// TIA Portal project "SistemaIrrigazione2" (V15.1)

(* hardware
DEVICE "S7-1200 station_1"  S7-1200 Station
   slot 0: "Telaio di montaggio_0"  S7-1200 Rack  Rack  V1.0
   slot 1: "PLC_1"  CPU 1214C DC/DC/DC  6ES7 214-1AG40-0XB0  V4.2
*)

// ===== PLC "PLC_1"  CPU 1214C DC/DC/DC =====

VAR_GLOBAL   // PLC tag table "Tabella delle variabili standard"
   "SEC" AT %I0.0 : Bool;
   "Apri_0" AT %Q0.1 : Bool;
   "Apri_1" AT %Q0.2 : Bool;
   "Apri_2" AT %Q0.3 : Bool;
   "Chiudi_0" AT %Q0.4 : Bool;
   "Chiudi_1" AT %Q0.5 : Bool;
   "Chiudi_2" AT %Q0.6 : Bool;
END_VAR

VAR_GLOBAL CONSTANT   // PLC tag table "Tabella delle variabili standard"
   "IntervalloIrrigazione" : Time := T#5m;
   "DurataApertura" : Time := T#10s;
   "DurataChiusura" : Time := T#10s;
   "DurataIrrigazioneRamo" : Time := T#40s;
END_VAR

TYPE "StructIrrigazioneRamo"
   STRUCT
      Home : Bool := true;
      Apertura : Bool;
      Irrigazione : Bool;
      Chiusura : Bool;
   END_STRUCT;
END_TYPE

DATA_BLOCK "IrrigazioneRamoFB_DB"   // DB1
{ S7_Optimized_Access := 'TRUE' }
VERSION : 0.1
// stored: InstanceOfName IrrigazioneRamoFB
"IrrigazioneRamoFB"
BEGIN
END_DATA_BLOCK

DATA_BLOCK "IrrigazioneRamoFB_DB_1"   // DB2
{ S7_Optimized_Access := 'TRUE' }
VERSION : 0.1
// stored: InstanceOfName IrrigazioneRamoFB
"IrrigazioneRamoFB"
BEGIN
END_DATA_BLOCK

DATA_BLOCK "IrrigazioneRamoFB_DB_2"   // DB5
{ S7_Optimized_Access := 'TRUE' }
VERSION : 0.1
// stored: InstanceOfName IrrigazioneRamoFB
"IrrigazioneRamoFB"
BEGIN
END_DATA_BLOCK

// folder: System blocks/Program resources

DATA_BLOCK "IEC_Timer_0_DB"   // DB3
{ S7_Optimized_Access := 'TRUE' }
AUTHOR : Simatic
FAMILY : IEC
NAME : IEC_TMR
VERSION : 1.0
// stored: InstanceOfName IEC_TIMER
"IEC_TIMER"
BEGIN
END_DATA_BLOCK

// folder: (top level)

FUNCTION_BLOCK "IrrigazioneRamoFB"   // FB1, LAD
{ S7_Optimized_Access := 'TRUE' }
VERSION : 0.1
   VAR_INPUT
      Abilita : Bool;
      DurataApertura : Time;
      DurataChiusura : Time;
      DurataIrrigazione : Time;
   END_VAR
   VAR_OUTPUT
      Apri : Bool;
      Chiudi : Bool;
   END_VAR
   VAR RETAIN
      IEC_Timer_0_Instance : TON_TIME;
      IEC_Timer_0_Instance_1 : TON_TIME;
      IEC_Timer_0_Instance_2 : TON_TIME;
      Stato : "StructIrrigazioneRamo";
   END_VAR
BEGIN

REGION Network 1
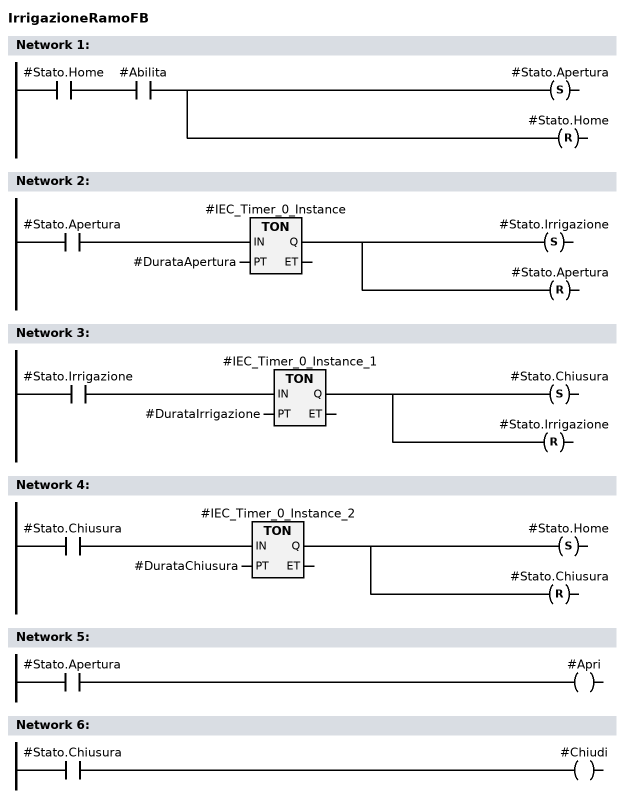
   RUNG wire#powerrail
      Contact( #Stato.Home )
      Contact( #Abilita )
      wire#w1
      S_Coil( #Stato.Apertura )
   END_RUNG
   RUNG wire#w1
      R_Coil( #Stato.Home )
   END_RUNG
   // the same network as SCL:
   IF #Stato.Home AND #Abilita THEN
       #Stato.Apertura := TRUE;
       #Stato.Home := FALSE;
   END_IF;
END_REGION

REGION Network 2
   #IEC_Timer_0_Instance(IN := #Stato.Apertura, PT := #DurataApertura);   // TON
   IF #IEC_Timer_0_Instance.Q THEN
       #Stato.Irrigazione := TRUE;
       #Stato.Apertura := FALSE;
   END_IF;
END_REGION

REGION Network 3
   #IEC_Timer_0_Instance_1(IN := #Stato.Irrigazione, PT := #DurataIrrigazione);   // TON
   IF #IEC_Timer_0_Instance_1.Q THEN
       #Stato.Chiusura := TRUE;
       #Stato.Irrigazione := FALSE;
   END_IF;
END_REGION

REGION Network 4
   #IEC_Timer_0_Instance_2(IN := #Stato.Chiusura, PT := #DurataChiusura);   // TON
   IF #IEC_Timer_0_Instance_2.Q THEN
       #Stato.Home := TRUE;
       #Stato.Chiusura := FALSE;
   END_IF;
END_REGION

REGION Network 5
   RUNG wire#powerrail
      Contact( #Stato.Apertura )
      Coil( #Apri )
   END_RUNG
   // the same network as SCL:
   #Apri := #Stato.Apertura;
END_REGION

REGION Network 6
   RUNG wire#powerrail
      Contact( #Stato.Chiusura )
      Coil( #Chiudi )
   END_RUNG
   // the same network as SCL:
   #Chiudi := #Stato.Chiusura;
END_REGION
END_FUNCTION_BLOCK

ORGANIZATION_BLOCK "Main"   // OB1, LAD, ProgramCycle
TITLE = "Main Program Sweep (Cycle)"
{ S7_Optimized_Access := 'TRUE' }
VERSION : 0.1
   VAR_INPUT
      Initial_Call : Bool;   // Initial call of this OB
      Remanence : Bool;   // =True, if remanent data are available
   END_VAR
BEGIN

REGION Network 1
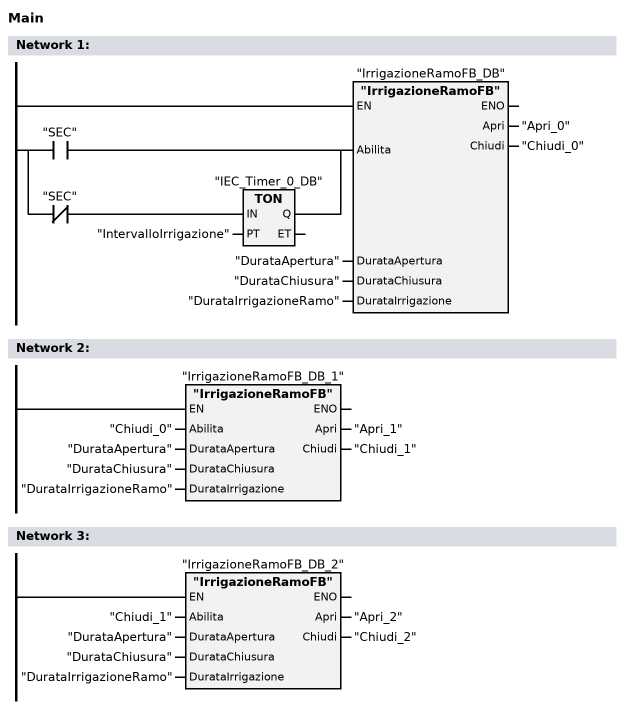
   "IEC_Timer_0_DB".TON(IN := NOT "SEC", PT := "IntervalloIrrigazione");
   "IrrigazioneRamoFB_DB"(Abilita := "SEC" OR "IEC_Timer_0_DB".Q,   // "IrrigazioneRamoFB"
                          DurataApertura := "DurataApertura",
                          DurataChiusura := "DurataChiusura",
                          DurataIrrigazione := "DurataIrrigazioneRamo",
                          Apri => "Apri_0",
                          Chiudi => "Chiudi_0");
END_REGION

REGION Network 2
   RUNG wire#powerrail
      "IrrigazioneRamoFB_DB_1"(Abilita := "Chiudi_0", DurataApertura := "DurataApertura", DurataChiusura := "DurataChiusura", DurataIrrigazione := "DurataIrrigazioneRamo", Apri => "Apri_1", Chiudi => "Chiudi_1")
   END_RUNG
   // the same network as SCL:
   "IrrigazioneRamoFB_DB_1"(Abilita := "Chiudi_0",   // "IrrigazioneRamoFB"
                           DurataApertura := "DurataApertura",
                           DurataChiusura := "DurataChiusura",
                           DurataIrrigazione := "DurataIrrigazioneRamo",
                           Apri => "Apri_1",
                           Chiudi => "Chiudi_1");
END_REGION

REGION Network 3
   RUNG wire#powerrail
      "IrrigazioneRamoFB_DB_2"(Abilita := "Chiudi_1", DurataApertura := "DurataApertura", DurataChiusura := "DurataChiusura", DurataIrrigazione := "DurataIrrigazioneRamo", Apri => "Apri_2", Chiudi => "Chiudi_2")
   END_RUNG
   // the same network as SCL:
   "IrrigazioneRamoFB_DB_2"(Abilita := "Chiudi_1",   // "IrrigazioneRamoFB"
                           DurataApertura := "DurataApertura",
                           DurataChiusura := "DurataChiusura",
                           DurataIrrigazione := "DurataIrrigazioneRamo",
                           Apri => "Apri_2",
                           Chiudi => "Chiudi_2");
END_REGION
END_ORGANIZATION_BLOCK